{attribute addProperty BoxType "EL2564-0000-0016"}
{attribute addProperty Id "StatusAT %I*Status_20B7064D162"}
{attribute addProperty CRC "903705316"}
{attribute addProperty SizeInBites "16"}
{attribute addProperty SizeInBytes "2"}
TYPE PWM_Inputs_Channel_35DD72E4 :
STRUCT
	{attribute addProperty Name "Status"}
	Status AT %I* : Status_20B7064D;
END_STRUCT
END_TYPE

(* stored: Version 1.2.0.0, ProductVersion 3.1.4024.9
   DUT PWM_Inputs_Channel_35DD72E4: Id {e39711b7-94c9-43c1-8ea3-f45a4f82f028} *)
